FUNCTION_BLOCK FB_HE_SATT_SequenceTestDouble IMPLEMENTS I_HE_SATT_Sequence
VAR
    fStartTransmissionValue : LREAL;
    eStartRoundingModeValue : E_HE_SATT_RoundingMode;
    fStartAllowableToleranceValue : LREAL;
END_VAR


METHOD PUBLIC GetStartAllowableToleranceValue : LREAL

GetStartAllowableToleranceValue := THIS^.fStartAllowableToleranceValue;
END_METHOD


METHOD PUBLIC GetStartRoundingModeValue : E_HE_SATT_RoundingMode

GetStartRoundingModeValue := THIS^.eStartRoundingModeValue;
END_METHOD


METHOD PUBLIC GetStartTransmissionValue : LREAL

GetStartTransmissionValue := THIS^.fStartTransmissionValue;
END_METHOD


METHOD Start
VAR_INPUT
    fRequestedTransmission : LREAL; // [0.0 - 1.0]
    eRequestedRoundingMode : E_HE_SATT_RoundingMode;
    fRequestedAllowableTolerance : LREAL;
END_VAR

THIS^.fStartTransmissionValue := fRequestedTransmission;
THIS^.eStartRoundingModeValue := eRequestedRoundingMode;
THIS^.fStartAllowableToleranceValue := fRequestedAllowableTolerance;
END_METHOD

END_FUNCTION_BLOCK

(* stored: Version 1.1.0.1
   POU FB_HE_SATT_SequenceTestDouble: Id {47db70f5-0512-48d8-9648-b9b46ca0ccce}, SpecialFunc None
   Method GetStartAllowableToleranceValue: Id {a3a67367-ac29-48e6-b6de-5afbbc2488a3}
   Method GetStartRoundingModeValue: Id {abcbc0f9-a20e-4e83-931d-25e446b8ab73}
   Method GetStartTransmissionValue: Id {e74118ec-f032-4530-8f94-664c658370ef}
   Method Start: Id {db9ed80d-6597-4a2c-9821-62df0218fc99} *)
